Omron CX-Programmer project NewProject (CX-Programmer 9.87)

# PLC NewPLC1: CP1L M

## Global symbols (name address type ; comment)
0.00 BOOL  ; Prensa 31
0.01 BOOL  ; Prensa 30
10.00 BOOL  ; auxiliar zeramento
10.01 BOOL  ; Inicio Turno 1 para transferir dados para BD
10.02 BOOL  ; Inicio Turno 2 para transferir dados para BD
10.03 BOOL  ; inicio Turno 3 pra transferir dados para BD
12.00 BOOL  ; zero minutos
12.01 BOOL  ; 20 minutos
12.02 BOOL  ; 40 minutos
20.00 BOOL  ; prensa 29 parada
21.00 BOOL  ; prensa 30 parada
22.00 BOOL  ; prensa 31 parada
A252 CHANNEL  ; ano clp
A253 CHANNEL  ; mes clp
A351 CHANNEL  ; min seg clp
A352 CHANNEL  ; hora e dia clp
A353 CHANNEL  ; mes e ano clp
A355 CHANNEL  ; hora clp
A356 CHANNEL  ; minuto clp
A357 CHANNEL  ; segundo clp
D100 CHANNEL  ; conta peças ph29
D102 CHANNEL  ; conta peças ph30
D104 CHANNEL  ; conta peças ph31
D205 CHANNEL  ; Segundos Relógio
D206 CHANNEL  ; Minutos Relógio
D207 CHANNEL  ; Horas Relogio
D208 CHANNEL  ; Dia Relógio
D209 CHANNEL  ; Mes Relogio
D210 CHANNEL  ; Ano Relógio
D211 CHANNEL  ; Ano Relógio 4 digitos
D290 CHANNEL  ; turno 1
D291 CHANNEL  ; turno 2
D292 CHANNEL  ; turno 3
D295 CHANNEL  ; string responsave turno
D296 CHANNEL  ; inicia a variavel responsável pelo tamanho dos dados que será salvo no banco
D297 CHANNEL  ; inicia a area de memoria salvar dados
D299 CHANNEL  ; ano 2 dig
D308 CHANNEL  ; bd conta peças ph 29
D309 CHANNEL  ; bd conta peças ph 30
D310 CHANNEL  ; bd conta peças ph 31
D319 CHANNEL  ; d320
D320 CHANNEL  ; ano bd
D321 CHANNEL  ; mes bd
D322 CHANNEL  ; dia bd
D323 CHANNEL  ; hora bd
D324 CHANNEL  ; minuto bd
D325 CHANNEL  ; seg bd
D327 CHANNEL  ; segundo bd
D350 CHANNEL  ; aux fim bd
D400 CHANNEL  ; dia do mes
D402 CHANNEL  ; pirmeiro DM de envio peças ph
D404 CHANNEL  ; Número cavidades na prensa31
D405 CHANNEL  ; Codigo do formato ph31
D406 CHANNEL  ; Número cavidades na prensa30
D407 CHANNEL  ; Codigo do formato ph30
D408 CHANNEL  ; Número cavidades na prensa29
D409 CHANNEL  ; Codigo do formato ph29
D410 CHANNEL  ; primeiro DM envio formato
D800 CHANNEL  ; horas
D802 CHANNEL  ; minutos
D804 CHANNEL  ; segundos
D806 CHANNEL  ; dia calendario
D808 CHANNEL  ; mes calendario
D810 CHANNEL  ; mês selecionado
D811 CHANNEL  ; linha selecionada
D910 CHANNEL  ; mês selecionado
H20.00 BOOL  ; Memória Atualiza Relogio pelo supervisório
H30.00 BOOL  ; inicia contagem turno 1
H30.01 BOOL  ; inicia contagem turno 2
H30.02 BOOL  ; iniio contagem turno 3
H30.04 BOOL  ; memoria de envio
H30.05 BOOL  ; retardo para fim do db
T0000 BOOL  ; retardo gravar bd
T0001 BOOL  ; Retardo ciclo da prensa
T0002 BOOL  ; Retardo ciclo da prensa
T0003 BOOL  ; Retardo ciclo da prensa
T0020 BOOL  ; filtro contagem peças
T0021 BOOL  ; filtro contagem peças
T0023 BOOL  ; filtro contagem peças
Banco_de_Dados_29 Contador_de_Peças_PH29
Banco_de_Dados_30 Contador_de_Peças_PH30
Banco_de_Dados_31 Contador_de_Peças_PH31
Conta_Peças Contador_de_Peças_PH31
HORA_DIA_CLP A352 CHANNEL  ; hora e dia clp
MES_ANO_CLP A353 CHANNEL  ; mes e ano clp
MIN_SEG_CLP A351 CHANNEL  ; minuto e segundo clp
PH11 0.03 BOOL
PH29 0.05 BOOL
PH30 0.04 BOOL
Visual_Formato_Trabalho_29 Formato_de_Trabalho_29
Visual_Formato_Trabalho_30 Formato_de_Trabalho_30
Visual_Formato_Trabalho_31 Formato_de_Trabalho_31
ano_2dig D294 CHANNEL  ; ano 2 dig auxiliar conversão ano 4 digitos
ano_bd D301 CHANNEL  ; ano bd
dia_bd D303 CHANNEL  ; dia bd
hora_bd D304 CHANNEL  ; hora bd
mes_bd D302 CHANNEL  ; mes bd
min_bd D305 CHANNEL  ; minuto bd
seg_bd D306 CHANNEL  ; seg bd
turno_bd D307 CHANNEL  ; turno para salvar no banco
xx Formato_de_Trabalho_29

## Program NuovoProgramma1 (cyclic task 0)
Local symbols
Codigo_Defeito1 D504 CHANNEL  ; codigo do defeito 1
Codigo_Defeito1_42 D524 CHANNEL  ; codigo do defeito 1
Codigo_Defeito1_43 D544 CHANNEL  ; codigo do defeito 1
Codigo_Defeito2 D505 CHANNEL  ; codigo do defeito 2
Codigo_Defeito2_42 D525 CHANNEL  ; codigo do defeito 2
Codigo_Defeito2_43 D545 CHANNEL  ; codigo do defeito 2
Codigo_Defeito3 D506 CHANNEL  ; codigo do defeito 3
Codigo_Defeito3_42 D526 CHANNEL  ; codigo do defeito 3
Codigo_Defeito3_43 D546 CHANNEL  ; codigo do defeito 3
F_31dias_vezes_2_ph30 D338 WORD
F_31dias_vezes_2_ph31 D330 WORD
F_Memoria_contagem_BCD_ph30 D344 WORD
F_Memoria_contagem_BCD_ph31 D336 WORD
F_Memória_de_Armazenagem_ph30 D342 WORD
F_Memória_de_Armazenagem_ph31 D334 WORD
F_Ponteiro_Dword_ph30 D340 WORD
F_Ponteiro_Dword_ph31 D332 WORD
KEEP 30.00 BOOL
MemAtuaReloSupervisorio H20.00 BOOL  ; Memória Atualiza Relogio pelo supervisório
Memoria_contagem_BCD_ph29 D328 WORD
Memoria_contagem_BCD_ph30 D518 WORD
Memoria_contagem_BCD_ph31 D308 WORD
Memoria_contagem_BIN_ph29 D326 WORD
Memoria_contagem_BIN_ph30 D516 WORD
Memoria_contagem_BIN_ph31 D306 WORD
Memória_de_Armazenagem_ph29 D324 WORD
Memória_de_Armazenagem_ph30 D314 WORD
Memória_de_Armazenagem_ph31 D304 WORD
PH13 0.02 BOOL  ; Prensa 29
PH29paradaT1 D1 CHANNEL  ; cnt prensa 31 parada T1
PH29paradaT2 D4 CHANNEL  ; cnt prensa 31 parada T2
PH29paradaT3 D7 CHANNEL  ; cnt prensa 31 parada T3
PH30paradaT1 D2 CHANNEL  ; cnt prensa 31 parada T1
PH30paradaT2 D5 CHANNEL  ; cnt prensa 31 parada T2
PH30paradaT3 D8 CHANNEL  ; cnt prensa 31 parada T3
PH31paradaT1 D3 CHANNEL  ; cnt prensa 31 parada T1
PH31paradaT2 D6 CHANNEL  ; cnt prensa 31 parada T2
PH31paradaT3 D9 CHANNEL  ; cnt prensa 31 parada T3
Ponteiro_Dword_ph29 D322 WORD
Ponteiro_Dword_ph30 D312 WORD
Ponteiro_Dword_ph31 D302 WORD
Qtde_Amostragem D507 CHANNEL  ; quantidade amostragem
Qtde_Amostragem_42 D527 CHANNEL  ; quantidade amostragem
Qtde_Amostragem_43 D547 CHANNEL  ; quantidade amostragem
Qualidade_Ano D508 CHANNEL  ; envio qualidade ano
Qualidade_Ano_42 D528 CHANNEL  ; envio qualidade ano
Qualidade_Ano_43 D548 CHANNEL  ; envio qualidade ano
Qualidade_Dia D510 CHANNEL  ; envio qualidade dia
Qualidade_Dia_42 D530 CHANNEL  ; envio qualidade dia
Qualidade_Dia_43 D550 CHANNEL  ; envio qualidade dia
Qualidade_Gatilho D500 CHANNEL  ; gatilho para ler qualidade
Qualidade_Gatilho_42 D520 CHANNEL  ; gatilho para ler qualidade
Qualidade_Gatilho_43 D540 CHANNEL  ; gatilho para ler qualidade
Qualidade_Hora D511 CHANNEL  ; envio qualidade hora
Qualidade_Hora_42 D531 CHANNEL  ; envio qualidade hora
Qualidade_Hora_43 D551 CHANNEL  ; envio qualidade hora
Qualidade_Maquina_Current D514 CHANNEL  ; qualidade maquina atual
Qualidade_Maquina_Current_42 D534 CHANNEL  ; qualidade maquina atual
Qualidade_Maquina_Current_43 D554 CHANNEL  ; qualidade maquina atual
Qualidade_Maquina_Persisted D515 CHANNEL  ; qualidade maquina persistir
Qualidade_Maquina_Persisted_42 D535 CHANNEL  ; qualidade maquina persistir
Qualidade_Maquina_Persisted_43 D555 CHANNEL  ; qualidade maquina persistir
Qualidade_Mes D509 CHANNEL  ; envio qualidade me
Qualidade_Mes_42 D529 CHANNEL  ; envio qualidade me
Qualidade_Mes_43 D549 CHANNEL  ; envio qualidade me
Qualidade_Min D512 CHANNEL  ; envio qualidade min
Qualidade_Min_42 D532 CHANNEL  ; envio qualidade min
Qualidade_Min_43 D552 CHANNEL  ; envio qualidade min
Qualidade_Seg D513 CHANNEL  ; envio qualidade seg
Qualidade_Seg_42 D533 CHANNEL  ; envio qualidade seg
Qualidade_Seg_43 D553 CHANNEL  ; envio qualidade seg
Total_Defeitos1 D501 CHANNEL  ; total defeitos 1
Total_Defeitos1_42 D521 CHANNEL  ; total defeitos 1
Total_Defeitos1_43 D541 CHANNEL  ; total defeitos 1
Total_Defeitos2 D502 CHANNEL  ; total defeitos 2
Total_Defeitos2_42 D522 CHANNEL  ; total defeitos 2
Total_Defeitos2_43 D542 CHANNEL  ; total defeitos 2
Total_Defeitos3 D503 CHANNEL  ; total defeitos 3
Total_Defeitos3_42 D523 CHANNEL  ; total defeitos 3
Total_Defeitos3_43 D543 CHANNEL  ; total defeitos 3
_31dias_vezes_2_ph29 D320 WORD
_31dias_vezes_2_ph30 D310 WORD
_31dias_vezes_2_ph31 D300 WORD
ano4dig D211 CHANNEL  ; Ano Relógio 4 digitos
anoRelogio D210 CHANNEL  ; Ano Relógio
codFormPH29 D409 CHANNEL  ; Codigo do formato ph29
codFormPH30 D407 CHANNEL  ; Codigo do formato ph30
codFormPH31 D405 CHANNEL  ; Codigo do formato ph31
delayCicloPrensa29 T0001 BOOL  ; Retardo ciclo da prensa
delayCicloPrensa30 T0002 BOOL  ; Retardo ciclo da prensa
delayCicloPrensa31 T0003 BOOL  ; Retardo ciclo da prensa
diaCalendario D806 CHANNEL  ; dia calendario
diaMes D400 CHANNEL  ; dia do mes
diaRelogio D208 CHANNEL  ; Dia Relógio
filtroCntPc29 T0020 BOOL  ; filtro contagem peças
filtroCntPc30 T0021 BOOL  ; filtro contagem peças
filtroCntPc31 T0023 BOOL  ; filtro contagem peças
firstDMenvioFormat D410 CHANNEL  ; primeiro DM envio formato
firstDMenvioPcPH D402 CHANNEL  ; pirmeiro DM de envio peças ph
horaRelogio D207 CHANNEL  ; Horas Relogio
horas D800 CHANNEL  ; horas
iniciaCntTurno1 H30.00 BOOL  ; inicia contagem turno 1
iniciaCntTurno2 H30.01 BOOL  ; inicia contagem turno 2
iniciaCntTurno3 H30.02 BOOL  ; iniio contagem turno 3
linhaSelect D811 CHANNEL  ; linha selecionada
mesCalendario D808 CHANNEL  ; mes calendario
mesRelogio D209 CHANNEL  ; Mes Relogio
mesSelecionado D810 CHANNEL  ; mês selecionado
mesSelect D910 CHANNEL  ; mês selecionado
minutos D802 CHANNEL  ; minutos
minutosRelogio D206 CHANNEL  ; Minutos Relógio
numberCavidPH29 D408 CHANNEL  ; Número cavidades na prensa29
numberCavidPH30 D406 CHANNEL  ; Número cavidades na prensa30
numberCavidPH31 D404 CHANNEL  ; Número cavidades na prensa31
pecaPH29 D100 CHANNEL  ; conta peças ph29
pecaPH30 D102 CHANNEL  ; conta peças ph30
pecaPH31 D104 CHANNEL  ; conta peças ph31
ph29parada 20.00 BOOL  ; prensa 29 parada
ph30parada 21.00 BOOL  ; prensa 30 parada
ph31parada 22.00 BOOL  ; prensa 31 parada
ponteiroBDph29 D328 WORD  ; ponteiro banco de dados PH 29
ponteiroBDph30 D318 CHANNEL  ; ponteiro em BCD para armazenar a contagem
ponteiroBDph31 D308 WORD  ; ponteiro banco de dados PH31
prensa29 0.02 BOOL  ; Prensa 29
prensa30 0.01 BOOL  ; Prensa 30
prensa31 0.00 BOOL  ; Prensa 31
segundos D804 CHANNEL  ; segundos
segundosRelogio D205 CHANNEL  ; Segundos Relógio

### Section Reset

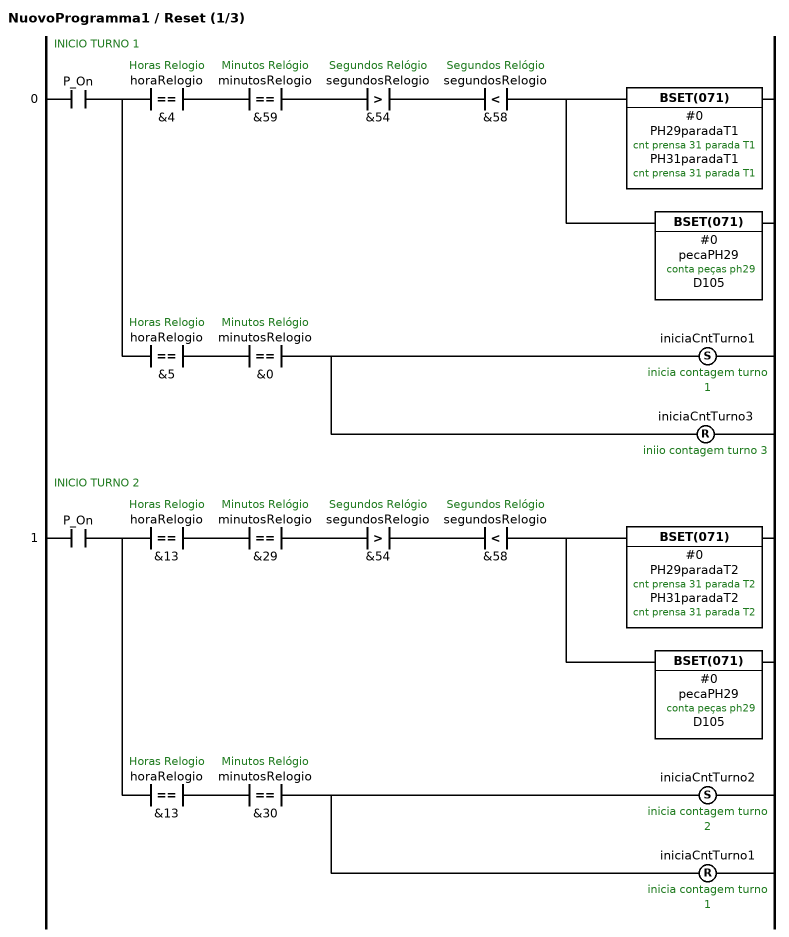
; rung 0: INICIO TURNO 1
LD P_On
OUT TR0
AND=(300) horaRelogio &4  ; Horas Relogio
AND=(300) minutosRelogio &59  ; Minutos Relógio
AND>(320) segundosRelogio &54  ; Segundos Relógio
AND<(310) segundosRelogio &58  ; Segundos Relógio
BSET(071) #0 PH29paradaT1 PH31paradaT1  ; cnt prensa 31 parada T1
BSET(071) #0 pecaPH29 D105  ; conta peças ph29
LD TR0
AND=(300) horaRelogio &5  ; Horas Relogio
AND=(300) minutosRelogio &0  ; Minutos Relógio
SET iniciaCntTurno1  ; inicia contagem turno 1
RSET iniciaCntTurno3  ; iniio contagem turno 3
; rung 1: INICIO TURNO 2
LD P_On
OUT TR0
AND=(300) horaRelogio &13  ; Horas Relogio
AND=(300) minutosRelogio &29  ; Minutos Relógio
AND>(320) segundosRelogio &54  ; Segundos Relógio
AND<(310) segundosRelogio &58  ; Segundos Relógio
BSET(071) #0 PH29paradaT2 PH31paradaT2  ; cnt prensa 31 parada T2
BSET(071) #0 pecaPH29 D105  ; conta peças ph29
LD TR0
AND=(300) horaRelogio &13  ; Horas Relogio
AND=(300) minutosRelogio &30  ; Minutos Relógio
SET iniciaCntTurno2  ; inicia contagem turno 2
RSET iniciaCntTurno1  ; inicia contagem turno 1

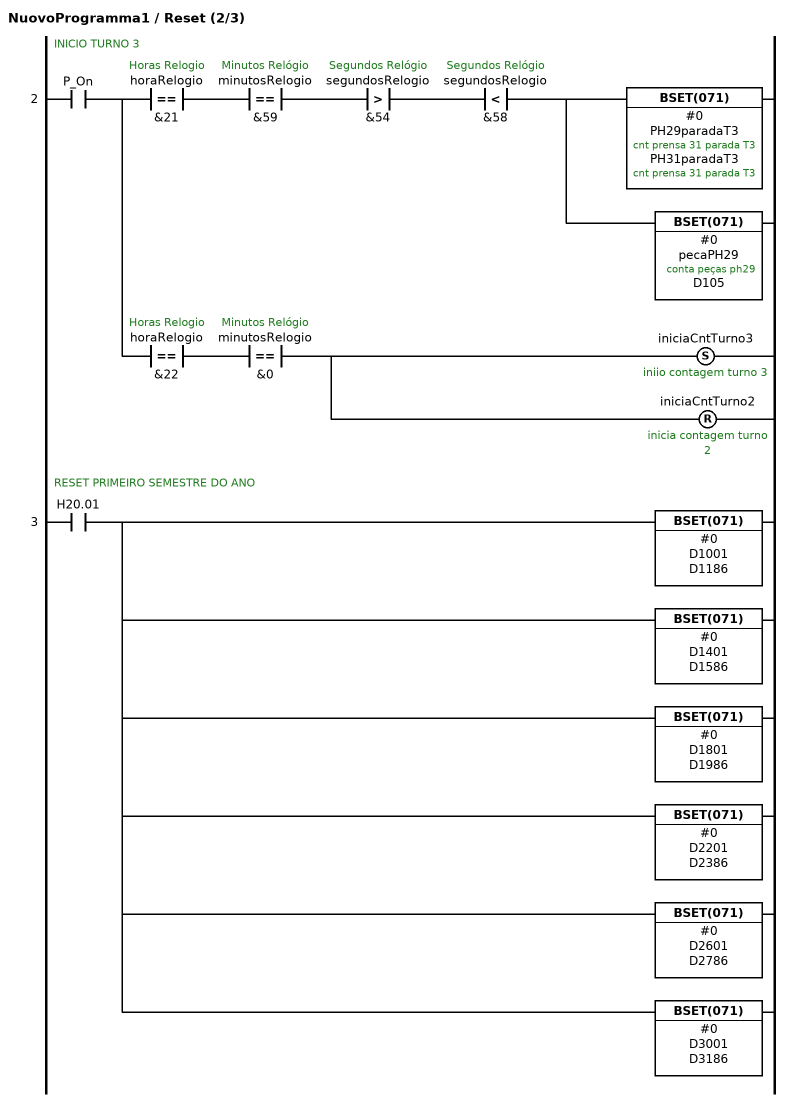
; rung 2: INICIO TURNO 3
LD P_On
OUT TR0
AND=(300) horaRelogio &21  ; Horas Relogio
AND=(300) minutosRelogio &59  ; Minutos Relógio
AND>(320) segundosRelogio &54  ; Segundos Relógio
AND<(310) segundosRelogio &58  ; Segundos Relógio
BSET(071) #0 PH29paradaT3 PH31paradaT3  ; cnt prensa 31 parada T3
BSET(071) #0 pecaPH29 D105  ; conta peças ph29
LD TR0
AND=(300) horaRelogio &22  ; Horas Relogio
AND=(300) minutosRelogio &0  ; Minutos Relógio
SET iniciaCntTurno3  ; iniio contagem turno 3
RSET iniciaCntTurno2  ; inicia contagem turno 2
; rung 3: RESET PRIMEIRO SEMESTRE DO ANO
LD H20.01
BSET(071) #0 D1001 D1186  // RESET PH31, 01/01 ATÉ 31/06
BSET(071) #0 D1401 D1586  // RESET PH30, 01/01 ATÉ 31/06
BSET(071) #0 D1801 D1986  // RESET PH29, 01/01 ATÉ 31/06
BSET(071) #0 D2201 D2386  // RESET FORMATO PH31, 01/01 ATÉ 31/06
BSET(071) #0 D2601 D2786  // RESET FORMATO PH30, 01/01 ATÉ 31/06
BSET(071) #0 D3001 D3186  // RESET FORMATO PH29, 01/01 ATÉ 31/06

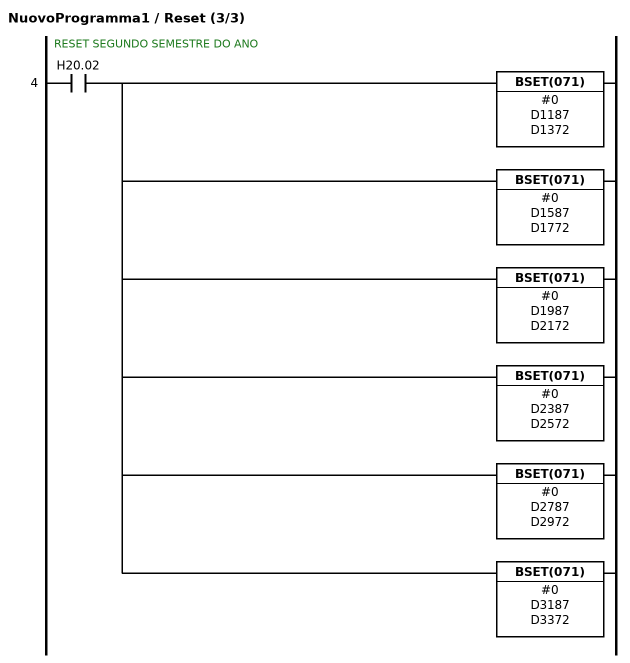
; rung 4: RESET SEGUNDO SEMESTRE DO ANO
LD H20.02
BSET(071) #0 D1187 D1372  // RESET PH31, 01/07 ATÉ 31/12
BSET(071) #0 D1587 D1772  // RESET PH30, 01/07 ATÉ 31/12
BSET(071) #0 D1987 D2172  // RESET PH29, 01/07 ATÉ 31/12
BSET(071) #0 D2387 D2572  // RESET FORMATO PH31, 01/07 ATÉ 31/12
BSET(071) #0 D2787 D2972  // RESET FORMATO PH30, 01/07 ATÉ 31/12
BSET(071) #0 D3187 D3372  // RESET FORMATO PH29, 01/07 ATÉ 31/12

### Section PH29

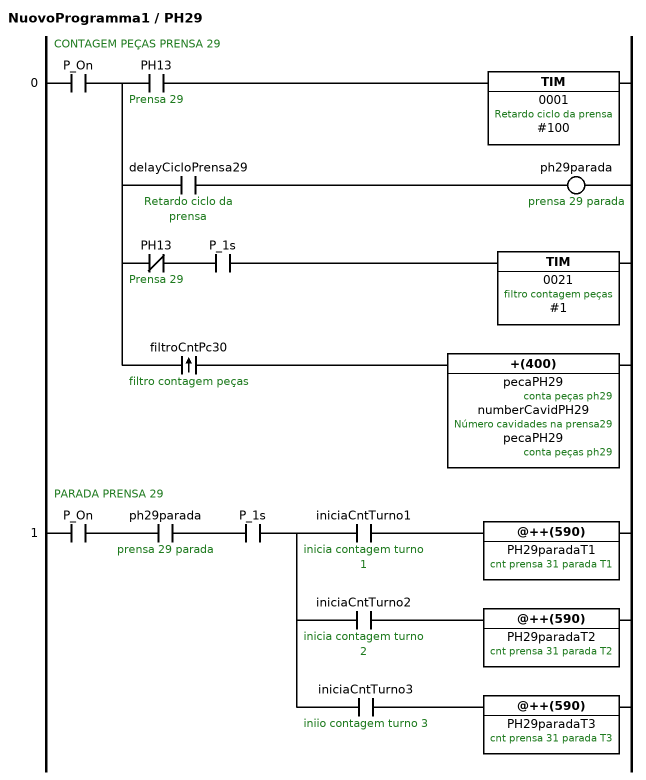
; rung 0: CONTAGEM PEÇAS PRENSA 29
LD P_On
OUT TR0
AND PH13  ; Prensa 29
TIM 0001 #100  ; Retardo ciclo da prensa
LD TR0
AND delayCicloPrensa29  ; Retardo ciclo da prensa
OUT ph29parada  ; prensa 29 parada
LD TR0
ANDNOT PH13  ; Prensa 29
AND P_1s
TIM 0021 #1  ; filtro contagem peças
LD TR0
@AND filtroCntPc30  ; filtro contagem peças
+(400) pecaPH29 numberCavidPH29 pecaPH29  ; conta peças ph29, Número cavidades na prensa29
; rung 1: PARADA PRENSA 29
LD P_On
AND ph29parada  ; prensa 29 parada
AND P_1s
OUT TR0
AND iniciaCntTurno1  ; inicia contagem turno 1
@++(590) PH29paradaT1  ; cnt prensa 31 parada T1  // CONTA PARADA TURNO 1
LD TR0
AND iniciaCntTurno2  ; inicia contagem turno 2
@++(590) PH29paradaT2  ; cnt prensa 31 parada T2  // CONTA PARADA TURNO 2
LD TR0
AND iniciaCntTurno3  ; iniio contagem turno 3
@++(590) PH29paradaT3  ; cnt prensa 31 parada T3  // CONTA PARADA TURNO 3

### Section PH30

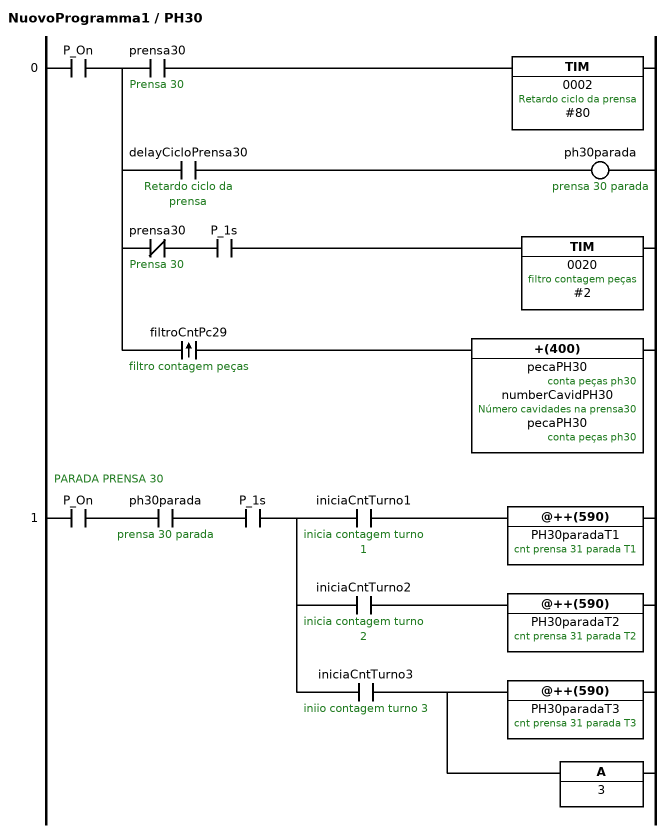
; rung 0
LD P_On
OUT TR0
AND prensa30  ; Prensa 30
TIM 0002 #80  ; Retardo ciclo da prensa
LD TR0
AND delayCicloPrensa30  ; Retardo ciclo da prensa
OUT ph30parada  ; prensa 30 parada
LD TR0
ANDNOT prensa30  ; Prensa 30
AND P_1s
TIM 0020 #2  ; filtro contagem peças
LD TR0
@AND filtroCntPc29  ; filtro contagem peças
+(400) pecaPH30 numberCavidPH30 pecaPH30  ; conta peças ph30, Número cavidades na prensa30
; rung 1: PARADA PRENSA 30
LD P_On  // D20 CONTA TURNO 2
AND ph30parada  ; prensa 30 parada
AND P_1s
OUT TR0
AND iniciaCntTurno1  ; inicia contagem turno 1
@++(590) PH30paradaT1  ; cnt prensa 31 parada T1  // 
LD TR0
AND iniciaCntTurno2  ; inicia contagem turno 2
@++(590) PH30paradaT2  ; cnt prensa 31 parada T2
LD TR0
AND iniciaCntTurno3  ; iniio contagem turno 3
@++(590) PH30paradaT3  ; cnt prensa 31 parada T3  // D18 CONTA TURNO 1
A  3
// D22 CONTA TURNO 3

### Section PH31

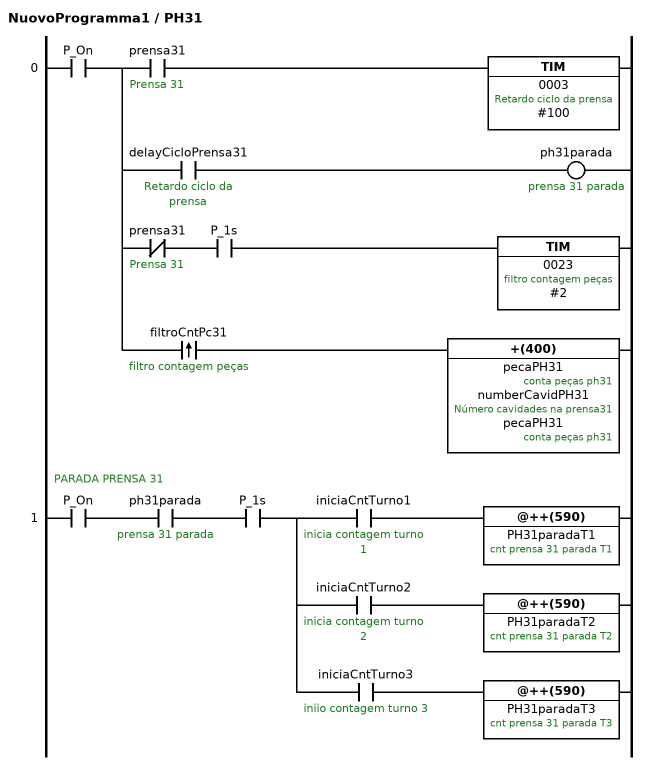
; rung 0
LD P_On
OUT TR0
AND prensa31  ; Prensa 31
TIM 0003 #100  ; Retardo ciclo da prensa
LD TR0
AND delayCicloPrensa31  ; Retardo ciclo da prensa
OUT ph31parada  ; prensa 31 parada
LD TR0
ANDNOT prensa31  ; Prensa 31
AND P_1s
TIM 0023 #2  ; filtro contagem peças
LD TR0
@AND filtroCntPc31  ; filtro contagem peças
+(400) pecaPH31 numberCavidPH31 pecaPH31  ; conta peças ph31, Número cavidades na prensa31
; rung 1: PARADA PRENSA 31
LD P_On
AND ph31parada  ; prensa 31 parada
AND P_1s
OUT TR0
AND iniciaCntTurno1  ; inicia contagem turno 1
@++(590) PH31paradaT1  ; cnt prensa 31 parada T1  // CONTA PARADA TURNO 1
LD TR0
AND iniciaCntTurno2  ; inicia contagem turno 2
@++(590) PH31paradaT2  ; cnt prensa 31 parada T2  // CONTA PARADA TURNO 2
LD TR0
AND iniciaCntTurno3  ; iniio contagem turno 3
@++(590) PH31paradaT3  ; cnt prensa 31 parada T3  // CONTA PARADA TUNOR 3

### Section Banco_de_Dados

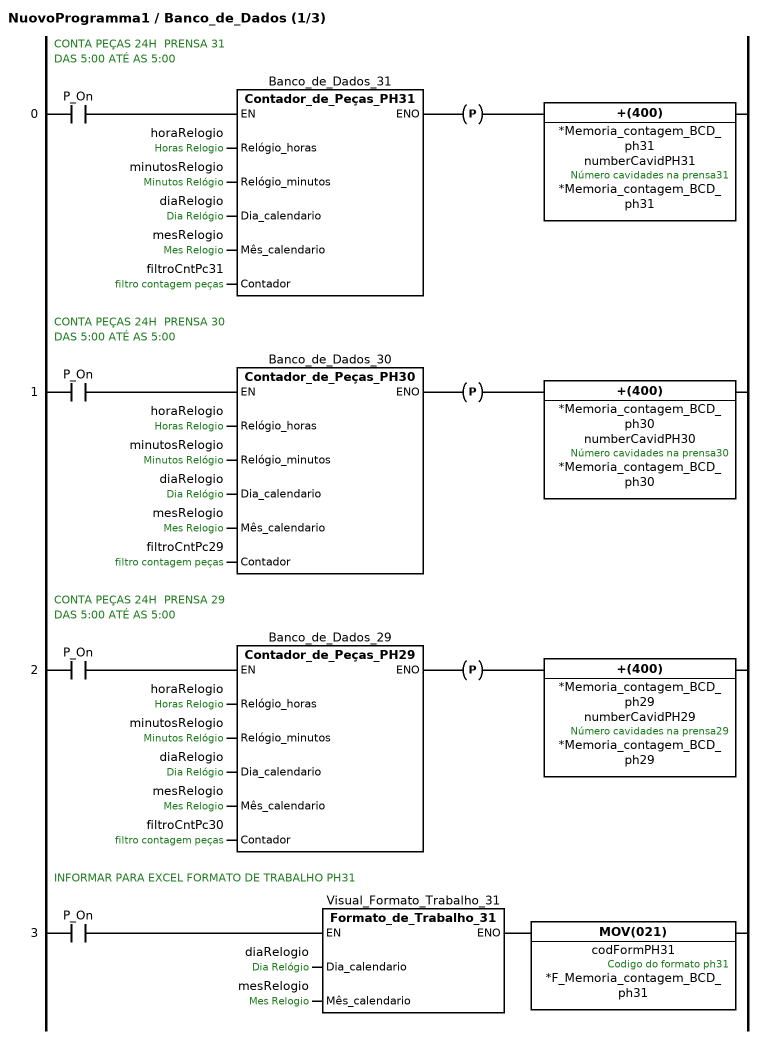
; rung 0: CONTA PEÇAS 24H  PRENSA 31 / DAS 5:00 ATÉ AS 5:00
LD P_On
CALL Banco_de_Dados_31 : Contador_de_Peças_PH31 (Relógio_horas := horaRelogio, Relógio_minutos := minutosRelogio, Dia_calendario := diaRelogio, Mês_calendario := mesRelogio, Contador := filtroCntPc31)  ; Horas Relogio, Minutos Relógio, Dia Relógio, Mes Relogio, filtro contagem peças
UP(521)
+(400) *Memoria_contagem_BCD_ph31 numberCavidPH31 *Memoria_contagem_BCD_ph31  ; Número cavidades na prensa31
; rung 1: CONTA PEÇAS 24H  PRENSA 30 / DAS 5:00 ATÉ AS 5:00
LD P_On
CALL Banco_de_Dados_30 : Contador_de_Peças_PH30 (Relógio_horas := horaRelogio, Relógio_minutos := minutosRelogio, Dia_calendario := diaRelogio, Mês_calendario := mesRelogio, Contador := filtroCntPc29)  ; Horas Relogio, Minutos Relógio, Dia Relógio, Mes Relogio, filtro contagem peças
UP(521)
+(400) *Memoria_contagem_BCD_ph30 numberCavidPH30 *Memoria_contagem_BCD_ph30  ; Número cavidades na prensa30
; rung 2: CONTA PEÇAS 24H  PRENSA 29 / DAS 5:00 ATÉ AS 5:00
LD P_On
CALL Banco_de_Dados_29 : Contador_de_Peças_PH29 (Relógio_horas := horaRelogio, Relógio_minutos := minutosRelogio, Dia_calendario := diaRelogio, Mês_calendario := mesRelogio, Contador := filtroCntPc30)  ; Horas Relogio, Minutos Relógio, Dia Relógio, Mes Relogio, filtro contagem peças
UP(521)
+(400) *Memoria_contagem_BCD_ph29 numberCavidPH29 *Memoria_contagem_BCD_ph29  ; Número cavidades na prensa29
; rung 3: INFORMAR PARA EXCEL FORMATO DE TRABALHO PH31
LD P_On
CALL Visual_Formato_Trabalho_31 : Formato_de_Trabalho_31 (Dia_calendario := diaRelogio, Mês_calendario := mesRelogio)  ; Dia Relógio, Mes Relogio
MOV(021) codFormPH31 *F_Memoria_contagem_BCD_ph31  ; Codigo do formato ph31

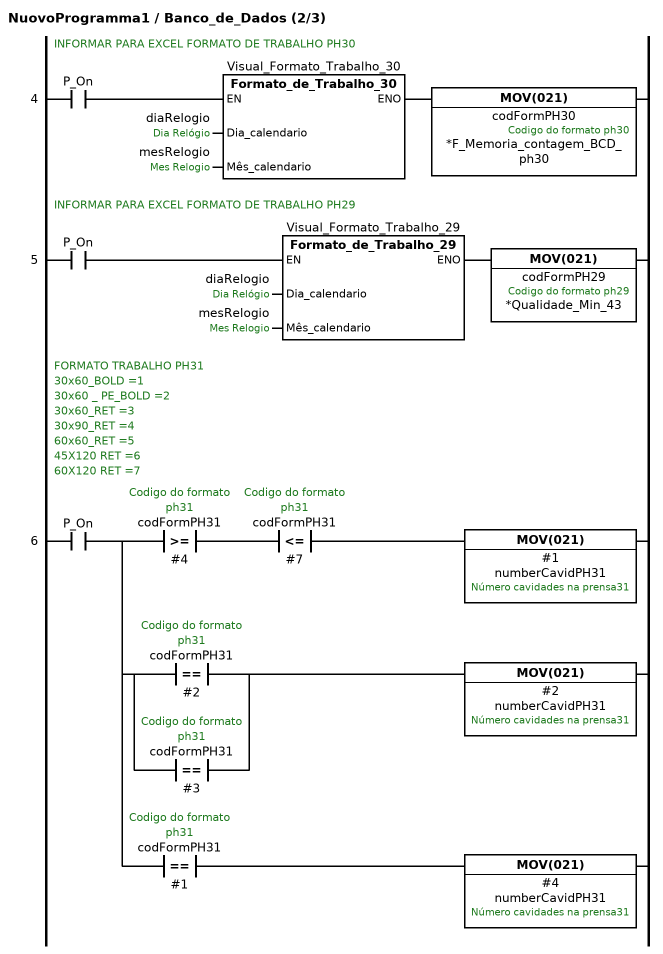
; rung 4: INFORMAR PARA EXCEL FORMATO DE TRABALHO PH30
LD P_On
CALL Visual_Formato_Trabalho_30 : Formato_de_Trabalho_30 (Dia_calendario := diaRelogio, Mês_calendario := mesRelogio)  ; Dia Relógio, Mes Relogio
MOV(021) codFormPH30 *F_Memoria_contagem_BCD_ph30  ; Codigo do formato ph30
; rung 5: INFORMAR PARA EXCEL FORMATO DE TRABALHO PH29
LD P_On
CALL Visual_Formato_Trabalho_29 : Formato_de_Trabalho_29 (Dia_calendario := diaRelogio, Mês_calendario := mesRelogio)  ; Dia Relógio, Mes Relogio
MOV(021) codFormPH29 *Qualidade_Min_43  ; Codigo do formato ph29
; rung 6: FORMATO TRABALHO PH31 / 30x60_BOLD =1 / 30x60_PE_BOLD =2 / 30x60_RET =3 / 30x90_RET =4 / 60x60_RET =5 / 45X120 RET =6 / 60X120 RET =7
LD P_On
OUT TR0
AND>=(325) codFormPH31 #4  ; Codigo do formato ph31
AND<=(315) codFormPH31 #7  ; Codigo do formato ph31
MOV(021) #1 numberCavidPH31  ; Número cavidades na prensa31
LD TR0
LD=(300) codFormPH31 #2  ; Codigo do formato ph31
OR=(300) codFormPH31 #3  ; Codigo do formato ph31
ANDLD
MOV(021) #2 numberCavidPH31  ; Número cavidades na prensa31
LD TR0
AND=(300) codFormPH31 #1  ; Codigo do formato ph31
MOV(021) #4 numberCavidPH31  ; Número cavidades na prensa31

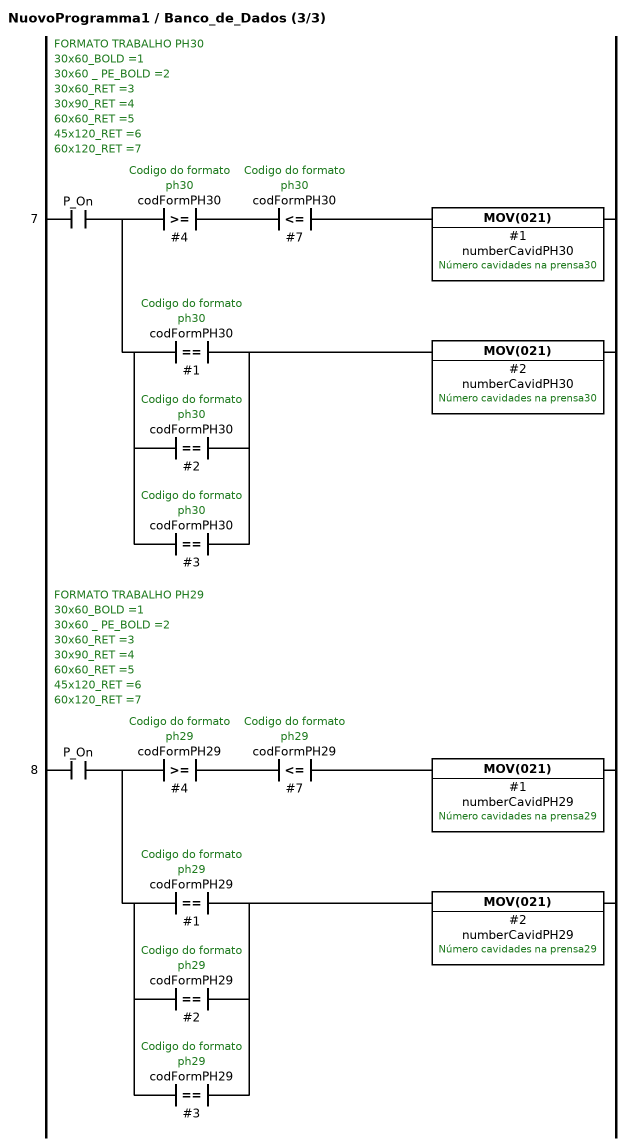
; rung 7: FORMATO TRABALHO PH30 / 30x60_BOLD =1 / 30x60_PE_BOLD =2 / 30x60_RET =3 / 30x90_RET =4 / 60x60_RET =5 / 45x120_RET =6 / 60x120_RET =7
LD P_On
OUT TR0
AND>=(325) codFormPH30 #4  ; Codigo do formato ph30
AND<=(315) codFormPH30 #7  ; Codigo do formato ph30
MOV(021) #1 numberCavidPH30  ; Número cavidades na prensa30
LD TR0
LD=(300) codFormPH30 #1  ; Codigo do formato ph30
OR=(300) codFormPH30 #2  ; Codigo do formato ph30
OR=(300) codFormPH30 #3  ; Codigo do formato ph30
ANDLD
MOV(021) #2 numberCavidPH30  ; Número cavidades na prensa30
; rung 8: FORMATO TRABALHO PH29 / 30x60_BOLD =1 / 30x60_PE_BOLD =2 / 30x60_RET =3 / 30x90_RET =4 / 60x60_RET =5 / 45x120_RET =6 / 60x120_RET =7
LD P_On
OUT TR0
AND>=(325) codFormPH29 #4  ; Codigo do formato ph29
AND<=(315) codFormPH29 #7  ; Codigo do formato ph29
MOV(021) #1 numberCavidPH29  ; Número cavidades na prensa29
LD TR0
LD=(300) codFormPH29 #1  ; Codigo do formato ph29
OR=(300) codFormPH29 #2  ; Codigo do formato ph29
OR=(300) codFormPH29 #3  ; Codigo do formato ph29
ANDLD
MOV(021) #2 numberCavidPH29  ; Número cavidades na prensa29

### Section Transferencia_excel

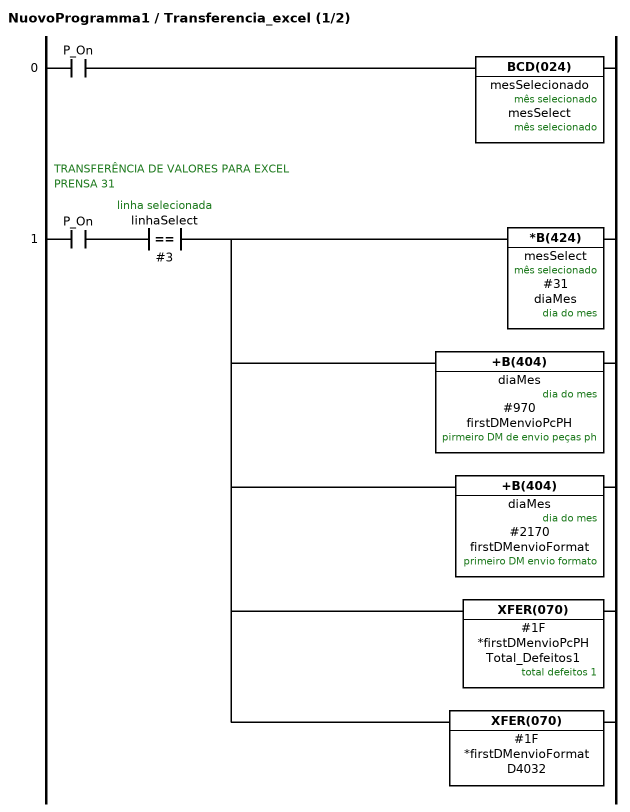
; rung 0
LD P_On
BCD(024) mesSelecionado mesSelect  ; mês selecionado
; rung 1: TRANSFERÊNCIA DE VALORES PARA EXCEL / PRENSA 31
LD P_On
AND=(300) linhaSelect #3  ; linha selecionada
*B(424) mesSelect #31 diaMes  ; mês selecionado, dia do mes
+B(404) diaMes #970 firstDMenvioPcPH  ; dia do mes, pirmeiro DM de envio peças ph
+B(404) diaMes #2170 firstDMenvioFormat  ; dia do mes, primeiro DM envio formato
XFER(070) #1F *firstDMenvioPcPH Total_Defeitos1  ; total defeitos 1
XFER(070) #1F *firstDMenvioFormat D4032

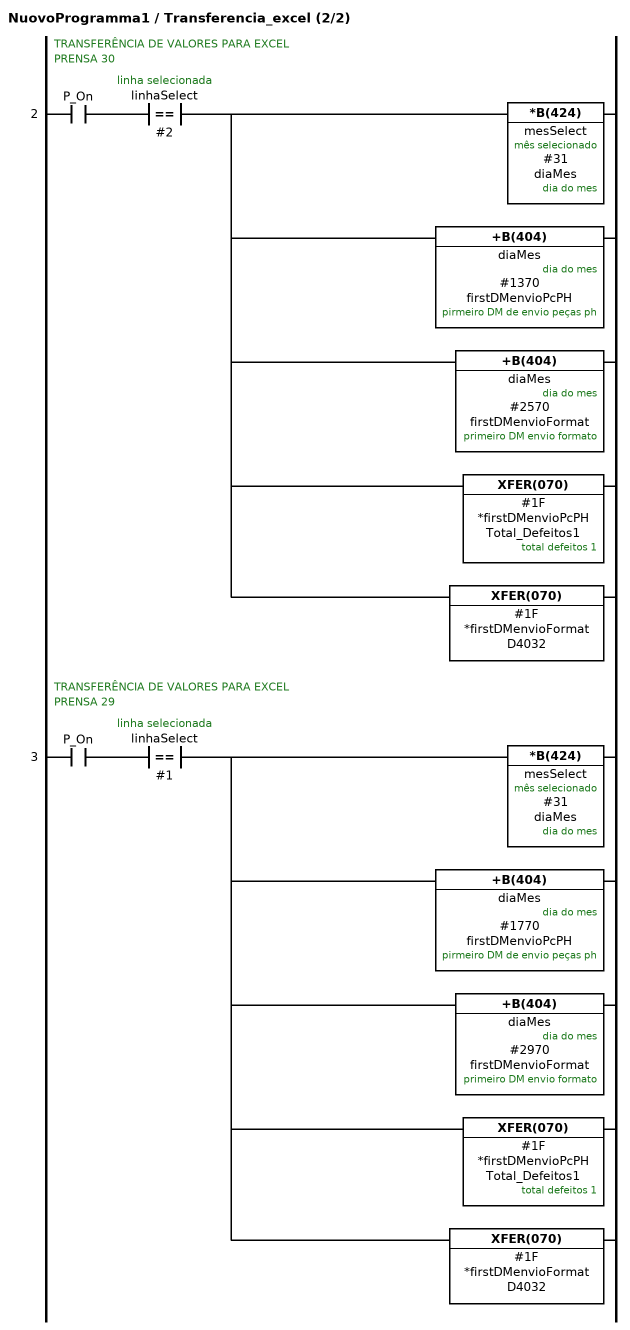
; rung 2: TRANSFERÊNCIA DE VALORES PARA EXCEL / PRENSA 30
LD P_On
AND=(300) linhaSelect #2  ; linha selecionada
*B(424) mesSelect #31 diaMes  ; mês selecionado, dia do mes
+B(404) diaMes #1370 firstDMenvioPcPH  ; dia do mes, pirmeiro DM de envio peças ph
+B(404) diaMes #2570 firstDMenvioFormat  ; dia do mes, primeiro DM envio formato
XFER(070) #1F *firstDMenvioPcPH Total_Defeitos1  ; total defeitos 1
XFER(070) #1F *firstDMenvioFormat D4032
; rung 3: TRANSFERÊNCIA DE VALORES PARA EXCEL / PRENSA 29
LD P_On
AND=(300) linhaSelect #1  ; linha selecionada
*B(424) mesSelect #31 diaMes  ; mês selecionado, dia do mes
+B(404) diaMes #1770 firstDMenvioPcPH  ; dia do mes, pirmeiro DM de envio peças ph
+B(404) diaMes #2970 firstDMenvioFormat  ; dia do mes, primeiro DM envio formato
XFER(070) #1F *firstDMenvioPcPH Total_Defeitos1  ; total defeitos 1
XFER(070) #1F *firstDMenvioFormat D4032

### Section Relogio

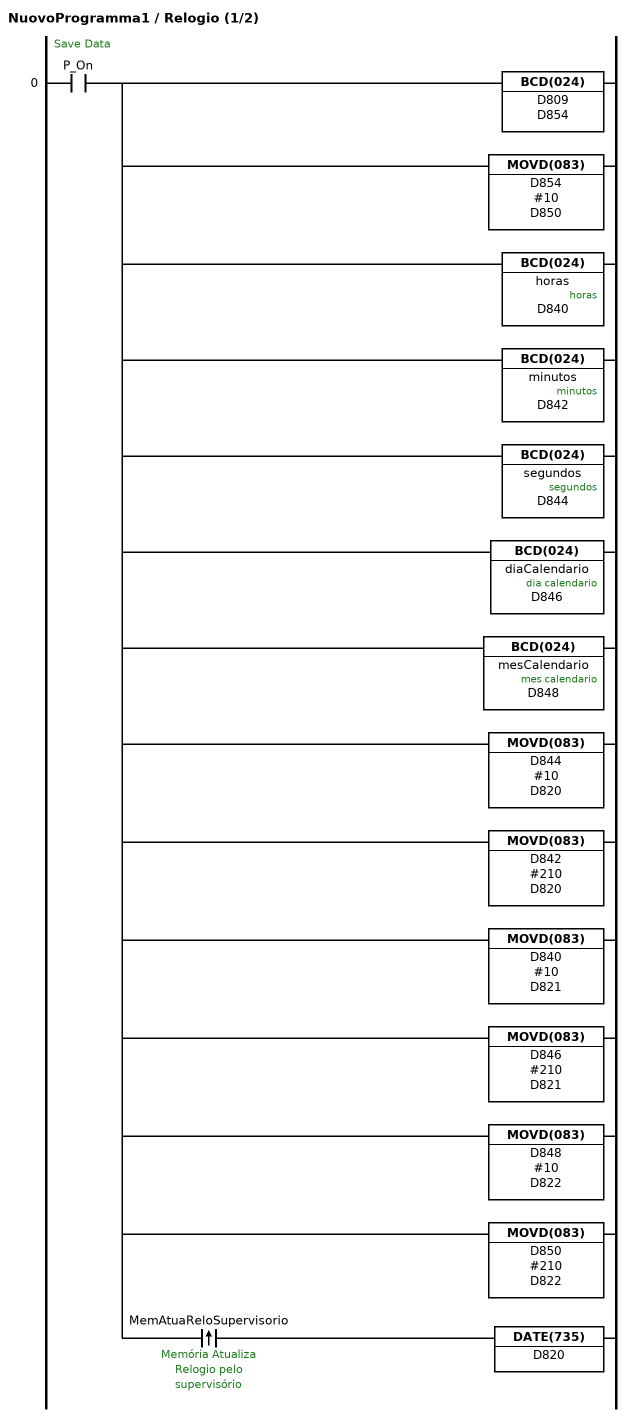
; rung 0: Save Data
LD P_On
BCD(024) D809 D854
MOVD(083) D854 #10 D850
BCD(024) horas D840  ; horas
BCD(024) minutos D842  ; minutos
BCD(024) segundos D844  ; segundos
BCD(024) diaCalendario D846  ; dia calendario
BCD(024) mesCalendario D848  ; mes calendario
MOVD(083) D844 #10 D820
MOVD(083) D842 #210 D820
MOVD(083) D840 #10 D821
MOVD(083) D846 #210 D821
MOVD(083) D848 #10 D822
MOVD(083) D850 #210 D822
@AND MemAtuaReloSupervisorio  ; Memória Atualiza Relogio pelo supervisório
DATE(735) D820

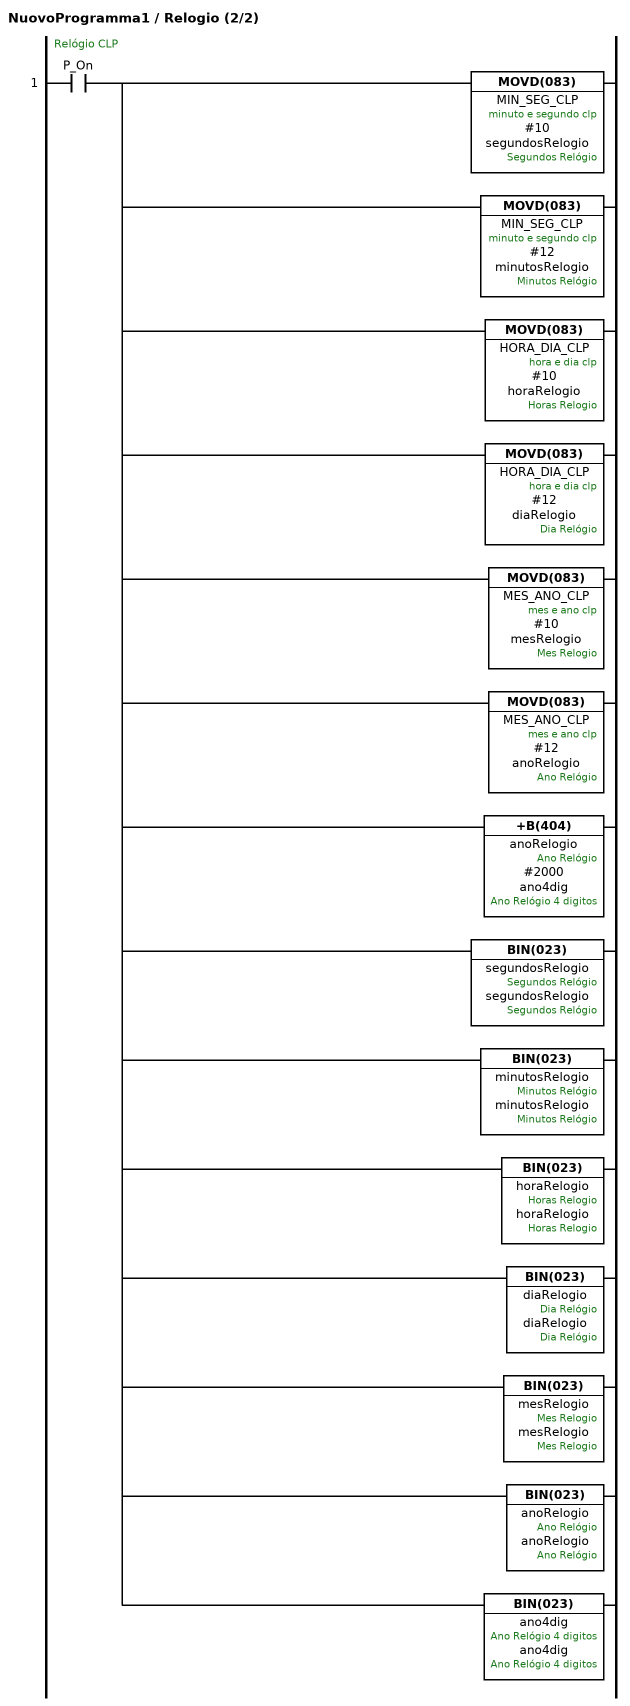
; rung 1: Relógio CLP
LD P_On
MOVD(083) MIN_SEG_CLP #10 segundosRelogio  ; minuto e segundo clp, Segundos Relógio
MOVD(083) MIN_SEG_CLP #12 minutosRelogio  ; minuto e segundo clp, Minutos Relógio
MOVD(083) HORA_DIA_CLP #10 horaRelogio  ; hora e dia clp, Horas Relogio
MOVD(083) HORA_DIA_CLP #12 diaRelogio  ; hora e dia clp, Dia Relógio
MOVD(083) MES_ANO_CLP #10 mesRelogio  ; mes e ano clp, Mes Relogio
MOVD(083) MES_ANO_CLP #12 anoRelogio  ; mes e ano clp, Ano Relógio
+B(404) anoRelogio #2000 ano4dig  ; Ano Relógio, Ano Relógio 4 digitos
BIN(023) segundosRelogio segundosRelogio  ; Segundos Relógio
BIN(023) minutosRelogio minutosRelogio  ; Minutos Relógio
BIN(023) horaRelogio horaRelogio  ; Horas Relogio
BIN(023) diaRelogio diaRelogio  ; Dia Relógio
BIN(023) mesRelogio mesRelogio  ; Mes Relogio
BIN(023) anoRelogio anoRelogio  ; Ano Relógio
BIN(023) ano4dig ano4dig  ; Ano Relógio 4 digitos

### Section ProducaoBD

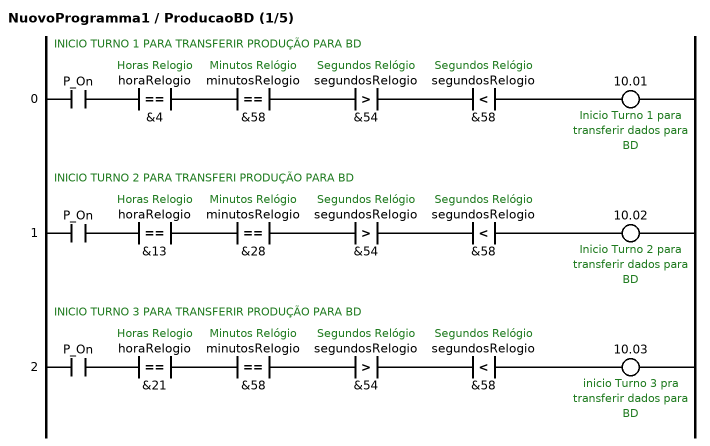
; rung 0: INICIO TURNO 1 PARA TRANSFERIR PRODUÇÃO PARA BD
LD P_On
AND=(300) horaRelogio &4  ; Horas Relogio
AND=(300) minutosRelogio &58  ; Minutos Relógio
AND>(320) segundosRelogio &54  ; Segundos Relógio
AND<(310) segundosRelogio &58  ; Segundos Relógio
OUT 10.01  ; Inicio Turno 1 para transferir dados para BD
; rung 1: INICIO TURNO 2 PARA TRANSFERI PRODUÇÃO PARA BD
LD P_On
AND=(300) horaRelogio &13  ; Horas Relogio
AND=(300) minutosRelogio &28  ; Minutos Relógio
AND>(320) segundosRelogio &54  ; Segundos Relógio
AND<(310) segundosRelogio &58  ; Segundos Relógio
OUT 10.02  ; Inicio Turno 2 para transferir dados para BD
; rung 2: INICIO TURNO 3 PARA TRANSFERIR PRODUÇÃO PARA BD
LD P_On
AND=(300) horaRelogio &21  ; Horas Relogio
AND=(300) minutosRelogio &58  ; Minutos Relógio
AND>(320) segundosRelogio &54  ; Segundos Relógio
AND<(310) segundosRelogio &58  ; Segundos Relógio
OUT 10.03  ; inicio Turno 3 pra transferir dados para BD

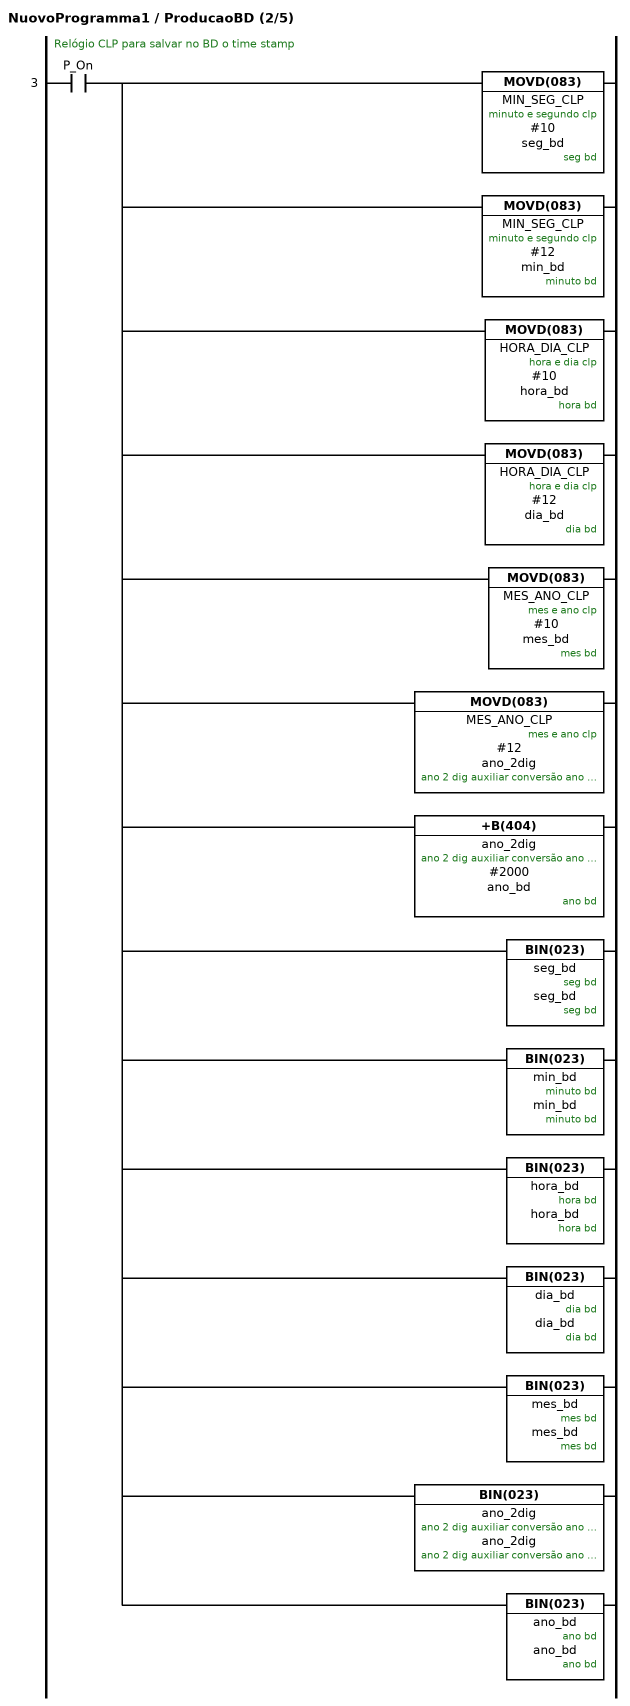
; rung 3: Relógio CLP para salvar no BD o time stamp
LD P_On
MOVD(083) MIN_SEG_CLP #10 seg_bd  ; minuto e segundo clp, seg bd
MOVD(083) MIN_SEG_CLP #12 min_bd  ; minuto e segundo clp, minuto bd
MOVD(083) HORA_DIA_CLP #10 hora_bd  ; hora e dia clp, hora bd
MOVD(083) HORA_DIA_CLP #12 dia_bd  ; hora e dia clp, dia bd
MOVD(083) MES_ANO_CLP #10 mes_bd  ; mes e ano clp, mes bd
MOVD(083) MES_ANO_CLP #12 ano_2dig  ; mes e ano clp, ano 2 dig auxiliar conversão ano 4 digitos
+B(404) ano_2dig #2000 ano_bd  ; ano 2 dig auxiliar conversão ano 4 digitos, ano bd
BIN(023) seg_bd seg_bd  ; seg bd
BIN(023) min_bd min_bd  ; minuto bd
BIN(023) hora_bd hora_bd  ; hora bd
BIN(023) dia_bd dia_bd  ; dia bd
BIN(023) mes_bd mes_bd  ; mes bd
BIN(023) ano_2dig ano_2dig  ; ano 2 dig auxiliar conversão ano 4 digitos
BIN(023) ano_bd ano_bd  ; ano bd

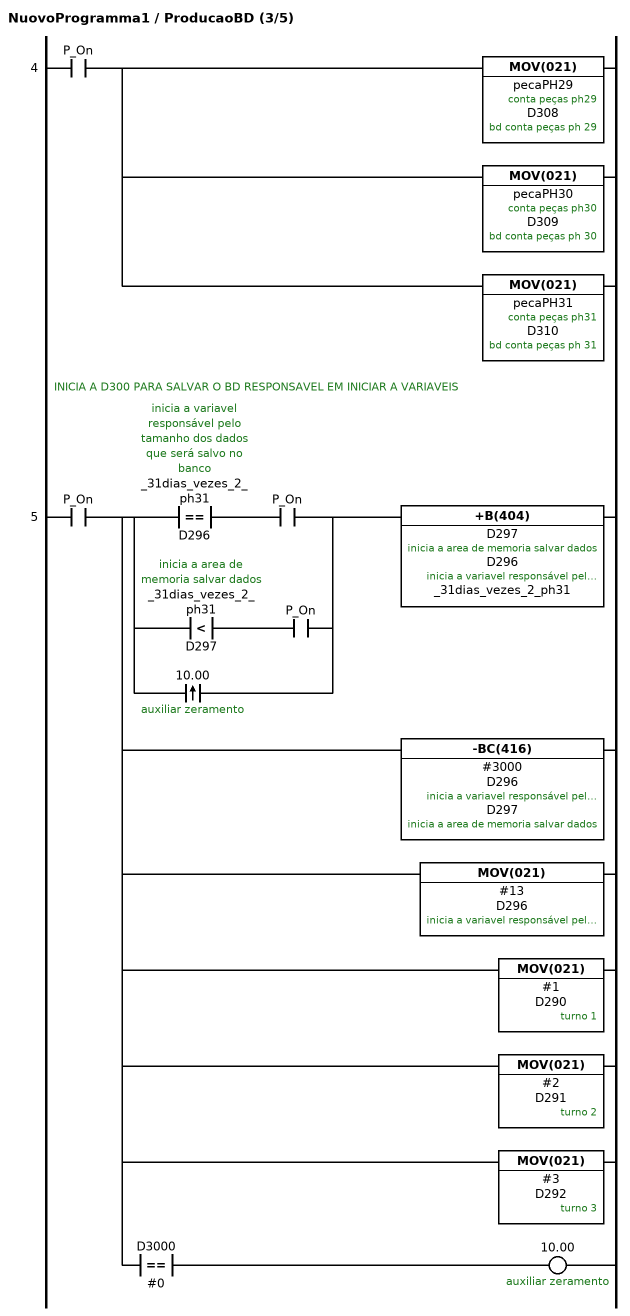
; rung 4
LD P_On
MOV(021) pecaPH29 D308  ; conta peças ph29, bd conta peças ph 29
MOV(021) pecaPH30 D309  ; conta peças ph30, bd conta peças ph 30
MOV(021) pecaPH31 D310  ; conta peças ph31, bd conta peças ph 31
; rung 5: INICIA A D300 PARA SALVAR O BD RESPONSAVEL EM INICIAR A VARIAVEIS
LD P_On
OUT TR0
LD=(300) _31dias_vezes_2_ph31 D296  ; inicia a variavel responsável pelo tamanho dos dados que será salvo no banco
AND P_On
LD<(310) _31dias_vezes_2_ph31 D297  ; inicia a area de memoria salvar dados
AND P_On
ORLD
@OR 10.00  ; auxiliar zeramento
ANDLD
+B(404) D297 D296 _31dias_vezes_2_ph31  ; inicia a area de memoria salvar dados, inicia a variavel responsável pelo tamanho dos dados que será salvo no banco  // inica a D300 ponteiro inicia responsál em salvar no banco
LD TR0
-BC(416) #3000 D296 D297  ; inicia a variavel responsável pelo tamanho dos dados que será salvo no banco, inicia a area de memoria salvar dados  // Inicia o endereço inicial para salvar no bd
MOV(021) #13 D296  ; inicia a variavel responsável pelo tamanho dos dados que será salvo no banco  // responsavel em determinar o tamanho do bd
MOV(021) #1 D290  ; turno 1  // inicia variavel turno 1
MOV(021) #2 D291  ; turno 2  // inicia variavel tuno 2
MOV(021) #3 D292  ; turno 3  // inicia a variavel turno 3
AND=(300) D3000 #0
OUT 10.00  ; auxiliar zeramento

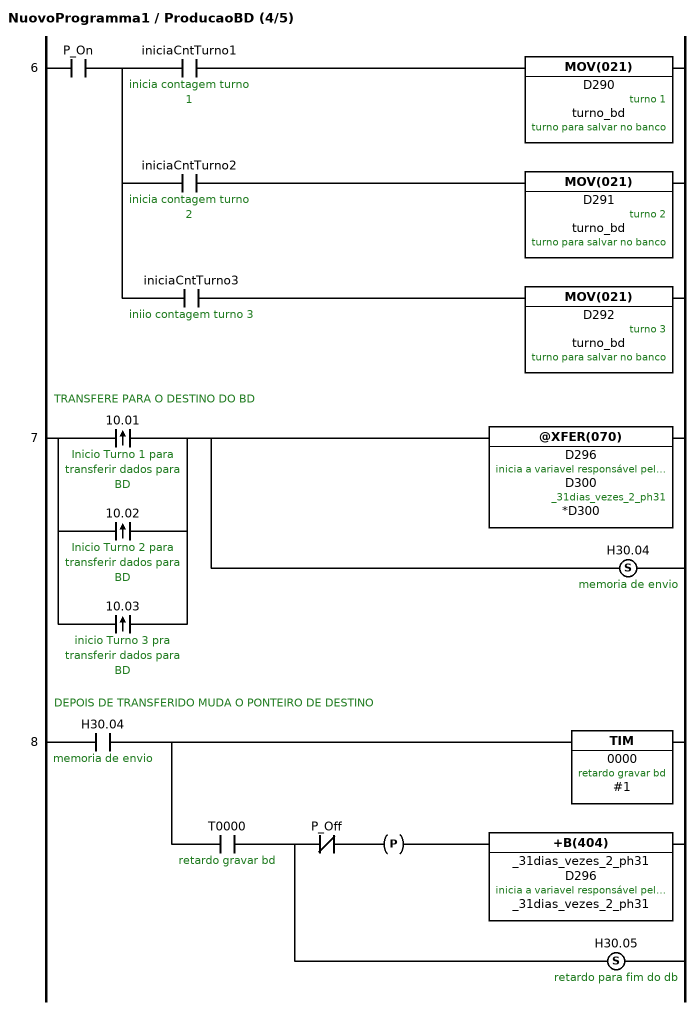
; rung 6
LD P_On
OUT TR0
AND iniciaCntTurno1  ; inicia contagem turno 1
MOV(021) D290 turno_bd  ; turno 1, turno para salvar no banco
LD TR0
AND iniciaCntTurno2  ; inicia contagem turno 2
MOV(021) D291 turno_bd  ; turno 2, turno para salvar no banco
LD TR0
AND iniciaCntTurno3  ; iniio contagem turno 3
MOV(021) D292 turno_bd  ; turno 3, turno para salvar no banco
; rung 7: TRANSFERE PARA O DESTINO DO BD
@LD 10.01  ; Inicio Turno 1 para transferir dados para BD
@OR 10.02  ; Inicio Turno 2 para transferir dados para BD
@OR 10.03  ; inicio Turno 3 pra transferir dados para BD
@XFER(070) D296 D300 *D300  ; inicia a variavel responsável pelo tamanho dos dados que será salvo no banco, _31dias_vezes_2_ph31
SET H30.04  ; memoria de envio
; rung 8: DEPOIS DE TRANSFERIDO MUDA O PONTEIRO DE DESTINO
LD H30.04  ; memoria de envio
TIM 0000 #1  ; retardo gravar bd
AND T0000  ; retardo gravar bd
OUT TR0
ANDNOT P_Off
UP(521)
+B(404) _31dias_vezes_2_ph31 D296 _31dias_vezes_2_ph31  ; inicia a variavel responsável pelo tamanho dos dados que será salvo no banco
LD TR0
SET H30.05  ; retardo para fim do db

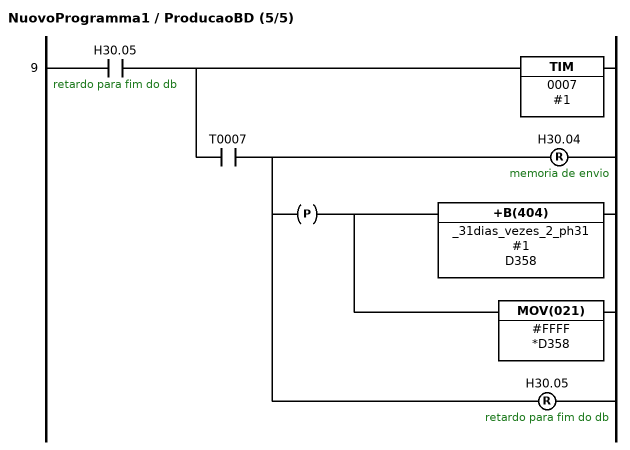
; rung 9
LD H30.05  ; retardo para fim do db
TIM 0007 #1
AND T0007
OUT TR0
RSET H30.04  ; memoria de envio
UP(521)
+B(404) _31dias_vezes_2_ph31 #1 D358
MOV(021) #FFFF *D358
LD TR0
RSET H30.05  ; retardo para fim do db

### Section QualidadeBD41

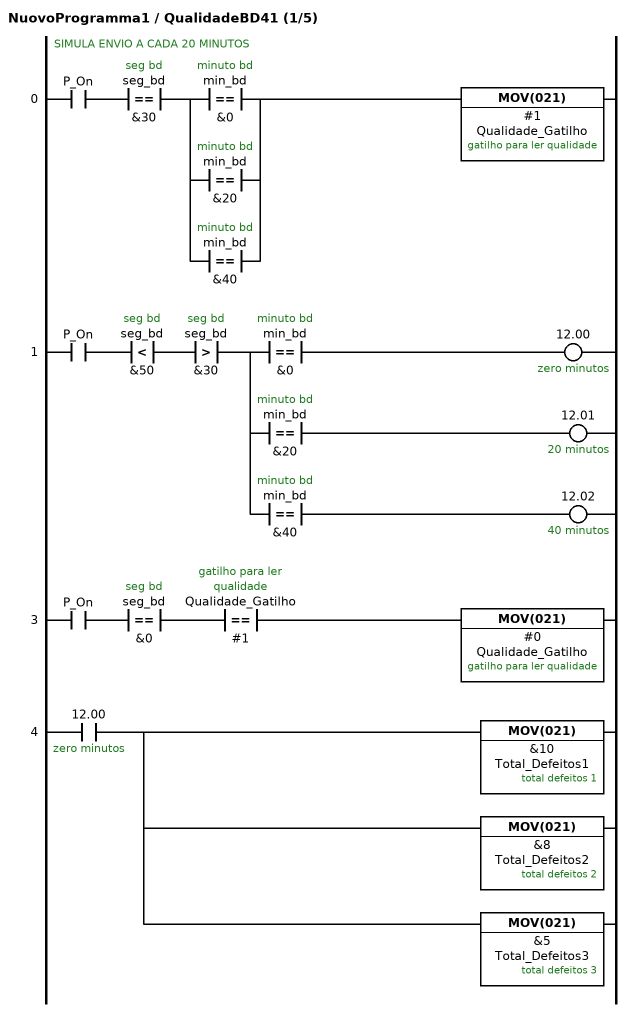
; rung 0: SIMULA ENVIO A CADA 20 MINUTOS
LD P_On
AND=(300) seg_bd &30  ; seg bd
LD=(300) min_bd &0  ; minuto bd
OR=(300) min_bd &20  ; minuto bd
OR=(300) min_bd &40  ; minuto bd
ANDLD
MOV(021) #1 Qualidade_Gatilho  ; gatilho para ler qualidade
; rung 1
LD P_On
AND<(310) seg_bd &50  ; seg bd
AND>(320) seg_bd &30  ; seg bd
OUT TR0
AND=(300) min_bd &0  ; minuto bd
OUT 12.00  ; zero minutos
LD TR0
AND=(300) min_bd &20  ; minuto bd
OUT 12.01  ; 20 minutos
LD TR0
AND=(300) min_bd &40  ; minuto bd
OUT 12.02  ; 40 minutos
; rung 3
LD P_On
AND=(300) seg_bd &0  ; seg bd
AND=(300) Qualidade_Gatilho #1  ; gatilho para ler qualidade
MOV(021) #0 Qualidade_Gatilho  ; gatilho para ler qualidade
; rung 4
LD 12.00  ; zero minutos
MOV(021) &10 Total_Defeitos1  ; total defeitos 1
MOV(021) &8 Total_Defeitos2  ; total defeitos 2
MOV(021) &5 Total_Defeitos3  ; total defeitos 3

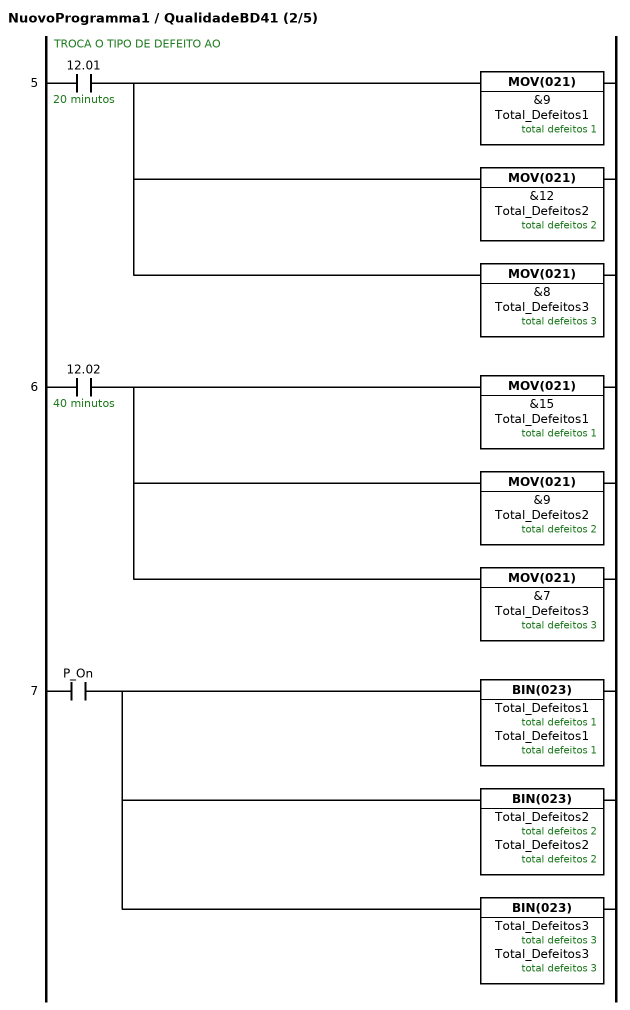
; rung 5: TROCA O TIPO DE DEFEITO AO
LD 12.01  ; 20 minutos
MOV(021) &9 Total_Defeitos1  ; total defeitos 1
MOV(021) &12 Total_Defeitos2  ; total defeitos 2
MOV(021) &8 Total_Defeitos3  ; total defeitos 3
; rung 6
LD 12.02  ; 40 minutos
MOV(021) &15 Total_Defeitos1  ; total defeitos 1
MOV(021) &9 Total_Defeitos2  ; total defeitos 2
MOV(021) &7 Total_Defeitos3  ; total defeitos 3
; rung 7
LD P_On
BIN(023) Total_Defeitos1 Total_Defeitos1  ; total defeitos 1
BIN(023) Total_Defeitos2 Total_Defeitos2  ; total defeitos 2
BIN(023) Total_Defeitos3 Total_Defeitos3  ; total defeitos 3

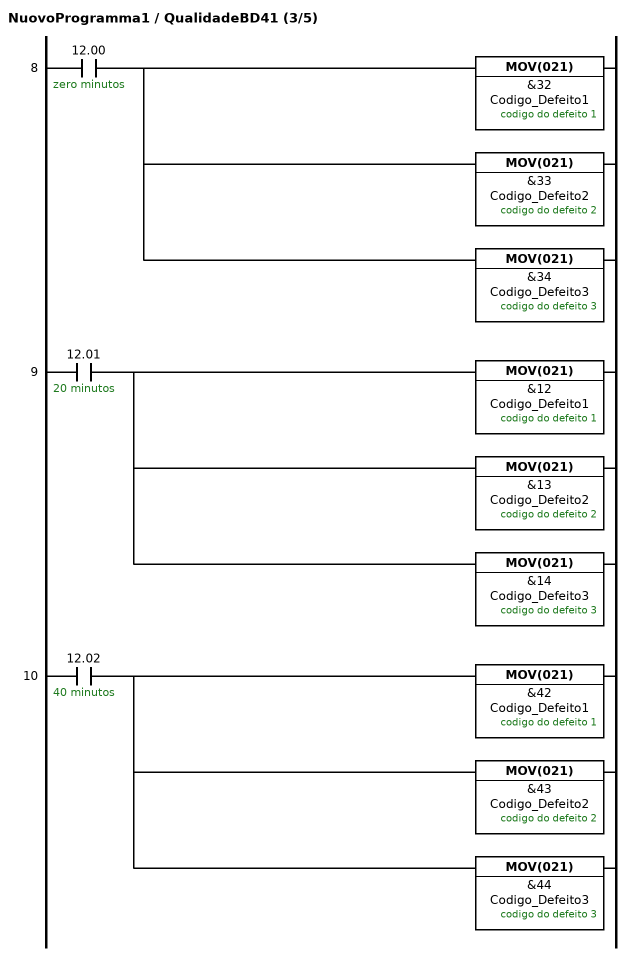
; rung 8
LD 12.00  ; zero minutos
MOV(021) &32 Codigo_Defeito1  ; codigo do defeito 1
MOV(021) &33 Codigo_Defeito2  ; codigo do defeito 2
MOV(021) &34 Codigo_Defeito3  ; codigo do defeito 3
; rung 9
LD 12.01  ; 20 minutos
MOV(021) &12 Codigo_Defeito1  ; codigo do defeito 1
MOV(021) &13 Codigo_Defeito2  ; codigo do defeito 2
MOV(021) &14 Codigo_Defeito3  ; codigo do defeito 3
; rung 10
LD 12.02  ; 40 minutos
MOV(021) &42 Codigo_Defeito1  ; codigo do defeito 1
MOV(021) &43 Codigo_Defeito2  ; codigo do defeito 2
MOV(021) &44 Codigo_Defeito3  ; codigo do defeito 3

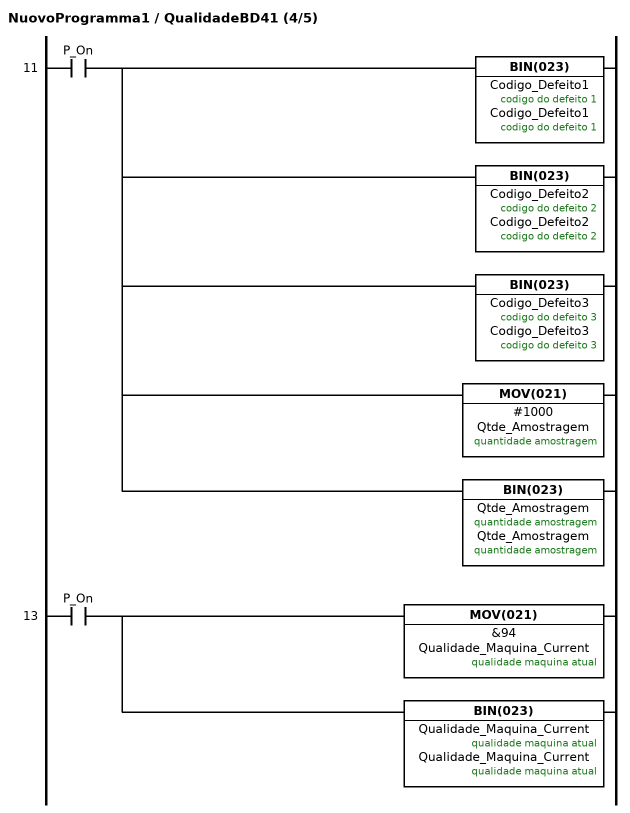
; rung 11
LD P_On
BIN(023) Codigo_Defeito1 Codigo_Defeito1  ; codigo do defeito 1
BIN(023) Codigo_Defeito2 Codigo_Defeito2  ; codigo do defeito 2
BIN(023) Codigo_Defeito3 Codigo_Defeito3  ; codigo do defeito 3
MOV(021) #1000 Qtde_Amostragem  ; quantidade amostragem
BIN(023) Qtde_Amostragem Qtde_Amostragem  ; quantidade amostragem
; rung 13
LD P_On
MOV(021) &94 Qualidade_Maquina_Current  ; qualidade maquina atual
BIN(023) Qualidade_Maquina_Current Qualidade_Maquina_Current  ; qualidade maquina atual

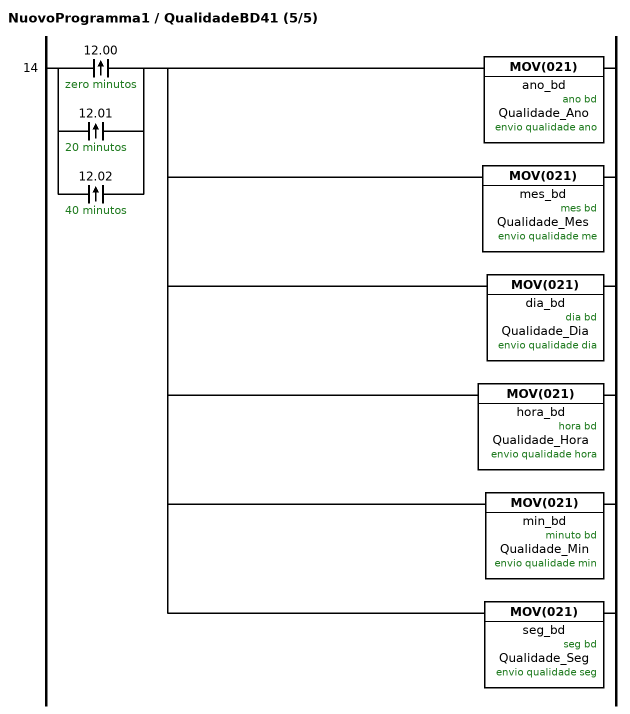
; rung 14
@LD 12.00  ; zero minutos
@OR 12.01  ; 20 minutos
@OR 12.02  ; 40 minutos
MOV(021) ano_bd Qualidade_Ano  ; ano bd, envio qualidade ano
MOV(021) mes_bd Qualidade_Mes  ; mes bd, envio qualidade me
MOV(021) dia_bd Qualidade_Dia  ; dia bd, envio qualidade dia
MOV(021) hora_bd Qualidade_Hora  ; hora bd, envio qualidade hora
MOV(021) min_bd Qualidade_Min  ; minuto bd, envio qualidade min
MOV(021) seg_bd Qualidade_Seg  ; seg bd, envio qualidade seg

### Section QualidadeBD42

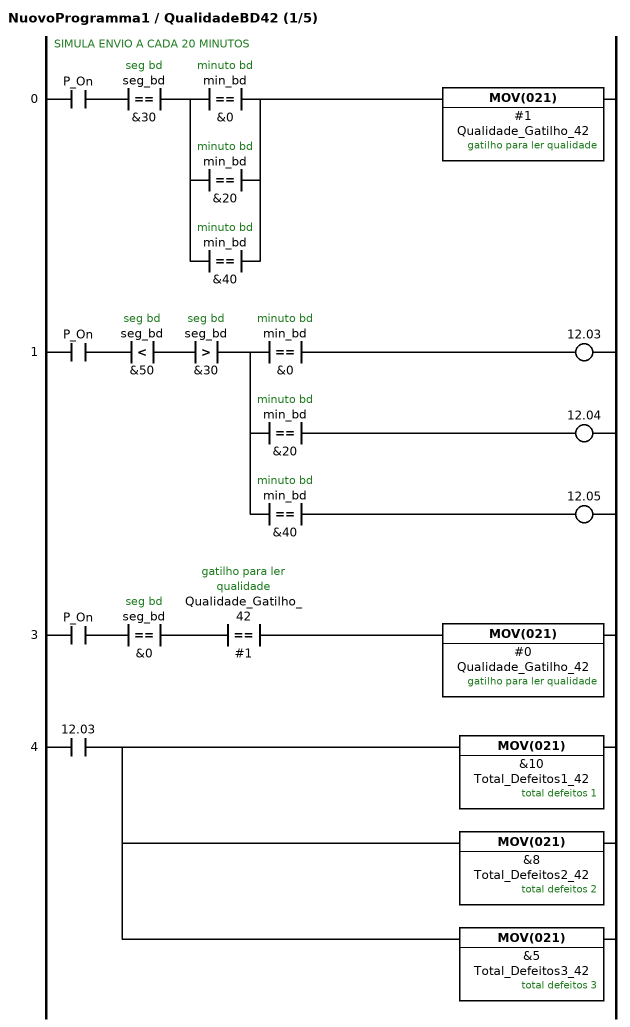
; rung 0: SIMULA ENVIO A CADA 20 MINUTOS
LD P_On
AND=(300) seg_bd &30  ; seg bd
LD=(300) min_bd &0  ; minuto bd
OR=(300) min_bd &20  ; minuto bd
OR=(300) min_bd &40  ; minuto bd
ANDLD
MOV(021) #1 Qualidade_Gatilho_42  ; gatilho para ler qualidade
; rung 1
LD P_On
AND<(310) seg_bd &50  ; seg bd
AND>(320) seg_bd &30  ; seg bd
OUT TR0
AND=(300) min_bd &0  ; minuto bd
OUT 12.03
LD TR0
AND=(300) min_bd &20  ; minuto bd
OUT 12.04
LD TR0
AND=(300) min_bd &40  ; minuto bd
OUT 12.05
; rung 3
LD P_On
AND=(300) seg_bd &0  ; seg bd
AND=(300) Qualidade_Gatilho_42 #1  ; gatilho para ler qualidade
MOV(021) #0 Qualidade_Gatilho_42  ; gatilho para ler qualidade
; rung 4
LD 12.03
MOV(021) &10 Total_Defeitos1_42  ; total defeitos 1
MOV(021) &8 Total_Defeitos2_42  ; total defeitos 2
MOV(021) &5 Total_Defeitos3_42  ; total defeitos 3

